TYPE EventText :
STRUCT
	event : I_TcEventBase;
	text  : REFERENCE TO STRING;
END_STRUCT
END_TYPE

(* stored: Version 1.1.0.1, ProductVersion 3.1.4024.15
   DUT EventText: Id {5cc6ca6e-1a7b-4282-90cd-b8e54235fe02} *)
